// TIA Portal V16 export
// export: Created 2022-11-17T15:49:37.0172366Z, ExportSetting WithDefaults, DisplayName Totally Integrated Automation Portal, DisplayVersion V16 Update 6, DisplayName TIA Portal Version Control Interface, DisplayVersion V16 Update 2, DisplayName TIA Portal Openness, DisplayVersion V16 Update 6, DisplayName SINAMICS Startdrive Advanced, DisplayVersion V16 Update 5, DisplayName SINAMICS Startdrive G130, G150, S120, S150, SINAMICS MV, S210, DisplayVersion V16 Update 5, DisplayName SINAMICS Startdrive G110M, G120, G120C, G120D, G120P, G115D, DisplayVersion V16 Update 5, DisplayName STEP 7 Professional, DisplayVersion V16 Update 6, DisplayName STEP 7 Safety, DisplayVersion V16, DisplayName WinCC Advanced, DisplayVersion V16 Update 6
DATA_BLOCK "DB07_TopAux"   // DB7
{ S7_Optimized_Access := 'FALSE' }
AUTHOR : Robopac
VERSION : 0.0
// stored: AutoNumber false, IsOnlyStoredInLoadMemory false, IsWriteProtectedInAS false
   VAR RETAIN
      VB700 : Byte := 16#00;
      V701_0 : Bool := TRUE;   // Top film is wrapped
      V701_1 : Bool := FALSE;   // Support memory for top wrapped
      V701_2 : Bool := FALSE;
      V701_3 : Bool := FALSE;
      V701_4 : Bool := FALSE;
      V701_5 : Bool := FALSE;
      V701_6 : Bool := FALSE;
      V701_7 : Bool := FALSE;
   END_VAR
BEGIN
END_DATA_BLOCK
